// TIA Portal V21 export
VAR_GLOBAL   // PLC tag table "K_Analogica"
END_VAR
VAR_GLOBAL CONSTANT   // user constants
   K_Analogica_LivelloVascaProdotto : Int := 1;   // Level tank product / Livello vasca prodotto
   K_Analogica_PressioneIngressoFiltriProdotto : Int := 2;   // Infeed product filter pressure / Pressione ingresso filtri prodotto
   K_Analogica_PressioneUscitaFiltriProdotto : Int := 3;   // Ausgangsdruck Produktfilter / Product filters outlet pressure / Presión de salida de los filtros del producto / Pression de sortie filtres produit / Pressione uscita filtri prodotto
   K_Analogica_PortataIngressoProdotto : Int := 4;   // DurchflussEingangProdukt / ProductInputRange / CaudalEntradaProducto / DébitEntréeProduit / PortataIngressoProdotto
   K_Analogica_PressioneSicurezzaIngressoSterilizzatore : Int := 5;   // Drucksicherheiteingangsterilisator / Pressuresafetysterilizerinput / Presiónseguridadentradaesterilizador / Pressionsécuritéentréestérilisateur / Pressionesicurezzaingressosterilizzatore
   K_Analogica_PressioneContropressioneIngressoPompaPistoni : Int := 6;   // Druck gegendruckeingangpumpekolben / Pressurebackpressurepistonpumpinlet / Presióncontrapresiónentradabombapistones / Pression contre-pressionentréepompepistons / Pressionecontropressioneingressopompapistoni
   K_Analogica_PressioneContropressioneFineLineaLavoro : Int := 7;   // Druck gegendruckendearbeitslinie / Pressurebackpressureworklineend / Presióncontrapresiónfinallíneatrabajo / Pression contre-pressionfinlignetravail / Pressionecontropressionefinelinealavoro
   K_Analogica_TemperaturaUscitaSterilizzatoreProcesso : Int := 8;   // Temperaturausgangsterilisatorprozess / Outputtemperaturesterilizerprocess / Temperaturasalidaesterilizadorproceso / Températuresortiestérilisateurprocessus / Temperaturauscitasterilizzatoreprocesso
   K_Analogica_TemperaturaAcquaCalda : Int := 9;   // Temperaturwassermantel / Warmwatertemperature / Temperaturaaguacalda / Températureeauchaud / Temperaturaacquacalda
   K_Analogica_TemperaturaIngressoSosta : Int := 10;   // Temperatureingangstopp / Stationinputtemperature / Temperaturaentradasosta / Températureentréestase / Temperaturaingressososta
   K_Analogica_TemperaturaUscitaSosta : Int := 11;   // Temperaturausgangstopp / Outputstoptemperature / Temperaturasalidasosta / Températuresortiestate / Temperaturauscitasosta
   K_Analogica_TemperaturaUscitaSterilizzatoreStoricizzare : Int := 12;   // Temperaturausgangsterilisatorstorization / Outputtemperaturesterilizerstoricize / Temperaturasalidaesterilizadorhistorizar / Températuresortiestérilisateurhistoriser / Temperaturauscitasterilizzatorestoricizzare
   K_Analogica_TemperaturaUscitaRaffredatoreProcesso : Int := 13;   // Temperaturausgangkühlerprozess / Outputtemperaturechillerprocess / Temperaturasalidarefrigeradorproceso / Température sortie refroidisseur processus / Temperaturauscitaraffredatoreprocesso
   K_Analogica_TemperaturaFineLinea : Int := 14;   // Temperaturlinienende / Lineendtemperature / Temperaturafinelínea / Températurefinligne / Temperaturafinelinea
   K_Analogica_TemperaturaBarriereVaporeValvScambio : Int := 15;   // Temperaturbarrierendampfvalvwechsel / Barriertemperaturevaporevalvexchange / Temperaturabarrerasvaporvalvintercambio / Températurebarrièrevapeurvalveéchange / Temperaturabarrierevaporevalvscambio
   K_Analogica_TemperaturaBarriereVaporeTuboInTubo : Int := 16;   // Temperaturbarrierendampfschlauchinschlauch / Barriertemperaturevaporetubeintube / Temperaturabarrerasvaportubointubo / Températurebarrièrevapeurtubeintube / Temperaturabarrierevaporetubointubo
   K_Analogica_TemperaturaUscitaSostaStoricizzazione : Int := 17;   // Temperaturausgangsteuerungstorisierung / Outputstockingstoricization temperature / Temperaturasalidasostahistorización / Températuresortiestathistorisation / Temperaturauscitasostastoricizzazione
   K_Analogica_TemperaturaRichiestaAcquaCalda : Int := 18;   // Temperaturanfragewassermantel / Warmwaterrequesttemperature / Temperaturasolicitudaguacalda / Températuredemandeeauchaud / Temperaturarichiestaacquacalda
   K_Analogica_LivelloSerbatoioCaldo : Int := 19;   // Füllstandbehälterkalk / Warmservoylevel / Niveldepósitocaldo / Niveauréservoirchaud / Livelloserbatoiocaldo
END_VAR
